PROGRAM MAIN_OOP
VAR
	bStartButton : PB_NOpen;
	bStopButton :PB_NOpen;
	bEstopButton : PB_NClose;
	bProcessStart : BOOL;
	bProcessError : BOOL;
	bProcessOverride : BOOL;
	
	//Feeder
	bStartFeeder		: BOOL;
	bStopFeeder			: BOOL;
	bFeederError        : BOOL;
	                   
	bFeederAuto         : BOOL;
	bFeederUpAuto       : BOOL;
	bFeederDownAuto     : BOOL;
	                   
	bFeederManual       : BOOL;
	bFeederUpManual     : BOOL;
	bFeederDownManual   : BOOL;
	
	bFeederAtPos		: BOOL;
	
	// SAT
	
	
END_VAR

IF bStartButton.IsPressed AND bStopButton.IsPressed THEN
	bStartFeeder:=TRUE;
END_IF
IF bStopButton.IsPressed AND bStartButton.IsPressed THEN
	bStopFeeder :=FALSE;
END_IF

P_MachineMain();

END_PROGRAM

(* stored: Version 1.1.0.1, ProductVersion 3.1.4024.12
   POU MAIN_OOP: Id {88f51528-a200-4dab-bc17-0a74643b910e}, SpecialFunc None *)
